// Mitsubishi GX Works2 project: CornCub   PLC: FX1S

// global labels: Global1
VAR_GLOBAL
  rHammerMill AT Y001 : BOOL;
  rMixer AT Y004 : BOOL;
  rLinear AT Y002 : BOOL;
  rPump AT Y000 : BOOL;
  rConveyor AT Y003 : BOOL;
  rHeater AT Y013 : BOOL;
  inStart AT X000 : BOOL;
  inStop AT X001 : BOOL;
  inHammerMill AT X002 : BOOL;
  inLinear AT X004 : BOOL;
  inMixer AT X003 : BOOL;
  inConveyor AT X005 : BOOL;
  inPump AT X006 : BOOL;
  inHeater AT X007 : BOOL;
  senEndConveyor AT X013 : BOOL;
  RunAutoFlag : BOOL;
  RunAutoStatus : INT;
  lStart AT Y007 : BOOL;
  lStop AT Y010 : BOOL;
  lTimerHammerMill AT Y011 : BOOL;
  lTimerMixer AT Y012 : BOOL;
  rTimerHammerMill AT Y005 : BOOL;
  rTimerMixer AT Y006 : BOOL;
  TimerHammerMillStat : BOOL;
  senTimerHammerMill AT X010 : BOOL;
END_VAR
VAR_GLOBAL CONSTANT
  blinkInterval : TIME := T#200ms;
END_VAR

// task Task_01 (event TRUE, interval 0, priority 31): POU_01

PROGRAM POU_01
VAR
  HammerMillManual : SinglePushButton;
  MixerManual : SinglePushButton;
  LinearManual : SinglePushButton;
  ConveyorManual : SinglePushButton;
  PumpManual : SinglePushButton;
  blinkStart : Blink;
END_VAR
 (*Button Start*)
IF	inStart = TRUE THEN
	IF RunAutoFlag = FALSE THEN
		RunAutoFlag:= TRUE;
		RunAutoStatus:=1;
	ELSE
		CASE RunAutoStatus OF
			1:
				(* Hammer Mill Run*)
				;
			2:
				(* Wait Command To Start Mixer *)
				;
			3:
				(* Mixer Run *)
				;
			4:
				(* Wait Command To Start Pouring *)
				;
			5:
				(*  Linear Open *)
				;
			6:
				(* Conveyor Run Until The end of Conveyor*)
				;
			7:
				(* Wait Command to Move to Press*)
				;
			8:
				(* Move To Press Then Timer*)
				;
			9:
				(* Wait Command to start Pump*)
				;
			10:
				(* Wait Command to stop Pump*)
				;
		END_CASE;
	END_IF;
END_IF;

IF	inStop= TRUE THEN
	RunAutoFlag:= FALSE;
	RunAutoStatus:=0;
	TimerHammerMillStat:=0;
	
	(* Stop All*)
	rHammerMill:=FALSE;
	rMixer:=FALSE;
	rLinear:=FALSE;
	rConveyor:=FALSE;
	rPump:=FALSE;
	lStart:=FALSE;
	rTimerHammerMill:=FALSE;
	rTimerMixer:=FALSE;
	lTimerHammerMill:=FALSE;
	lTimerMixer:=FALSE;
	
END_IF;

IF RunAutoFlag = TRUE THEN
	lStop:= FALSE;
ELSE
	lStop:= TRUE;
END_IF;

IF RunAutoFlag = TRUE THEN
	CASE RunAutoStatus OF
			1:
				(* Hammer Mill Run*)
				
				rTimerHammerMill:=TRUE;
				rHammerMill:= TRUE;
				IF senTimerHammerMill = TRUE  AND TimerHammerMillStat = FALSE THEN
					TimerHammerMillStat := TRUE;
				END_IF;
				
				IF inHammerMill = TRUE AND TimerHammerMillStat = TRUE THEN
					TimerHammerMillStat := FALSE;
					rTimerHammerMill:=FALSE;
					rHammerMill:=FALSE;
					RunAutoStatus:= 2;
				END_IF;
				
				IF senTimerHammerMill = FALSE AND TimerHammerMillStat = TRUE THEN
					TimerHammerMillStat := FALSE;
					rTimerHammerMill:=FALSE;
					rHammerMill:=FALSE;
					RunAutoStatus:= 2;
				END_IF;
				blinkStart(Input:= TRUE ,Output:= lStart ,IntervalTime:= blinkInterval);
			2:
				(* Wait Command To Start Mixer *)
				;
			3:
				(* Mixer Run *)
				;
			4:
				(* Wait Command To Start Pouring *)
				;
			5:
				(*  Linear Open *)
				;
			6:
				(* Conveyor Run Until The end of Conveyor*)
				;
			7:
				(* Wait Command to Move to Press*)
				;
			8:
				(* Move To Press Then Timer*)
				;
			9:
				(* Wait Command to start Pump*)
				;
			10:
				(* Wait Command to stop Pump*)
				;
	END_CASE;
ELSE
	(* Manual Run *)
	HammerMillManual(btnInput:= inHammerMill ,output:= rHammerMill );
	MixerManual(btnInput:= inMixer ,output:= rMixer );
	LinearManual(btnInput:= inLinear ,output:= rLinear );
	ConveyorManual(btnInput:= inConveyor,output:= rConveyor );
	PumpManual(btnInput:= inPump ,output:= rPump );
	
	(* Heater Manual Run *)
	IF inHeater= TRUE THEN
		rHeater:= TRUE;
	ELSE
		rHeater:= FALSE;
	END_IF;
	
END_IF;
END_PROGRAM

FUNCTION_BLOCK Blink
VAR_INPUT
  Input : BOOL;
END_VAR
VAR_OUTPUT
  Output : BOOL;
END_VAR
VAR
  Memory : BOOL;
  OnTimer : TON;
END_VAR
VAR_INPUT
  IntervalTime : TIME;
END_VAR
VAR
  OffTimer : TON;
  PtTimer1 : TIME;
  PtTimer2 : TIME;
  TimeOff : TOF;
END_VAR
(* structured ladder/FBD written out as ST: instructions are called as NAME(EN, inputs, outputs); _pN, _eN, _tN stand for wires *)
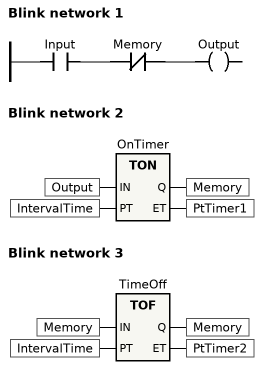
(* network 1 *)
Output := Input AND NOT Memory;
(* network 2 *)
OnTimer(IN := Output, PT := IntervalTime, Q => Memory, ET => PtTimer1);
(* network 3 *)
TimeOff(IN := Memory, PT := IntervalTime, Q => Memory, ET => PtTimer2);
END_FUNCTION_BLOCK

FUNCTION_BLOCK SinglePushButton
VAR_INPUT
  btnInput : BOOL;
END_VAR
VAR
  memoryOn : BOOL;
  memoryOff : BOOL;
END_VAR
VAR_OUTPUT
  output : BOOL;
END_VAR
(* structured ladder/FBD written out as ST: instructions are called as NAME(EN, inputs, outputs); _pN, _eN, _tN stand for wires *)
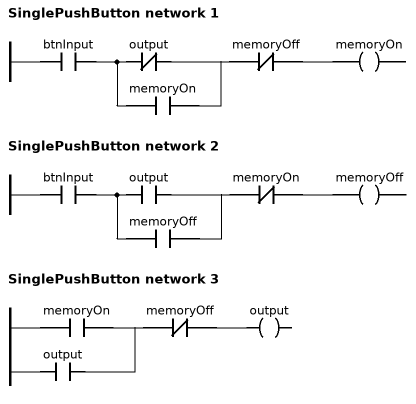
(* network 1 *)
memoryOn := ((btnInput AND NOT output) OR (btnInput AND memoryOn)) AND NOT memoryOff;
(* network 2 *)
memoryOff := ((btnInput AND output) OR (btnInput AND memoryOff)) AND NOT memoryOn;
(* network 3 *)
output := (memoryOn OR output) AND NOT memoryOff;
END_FUNCTION_BLOCK
